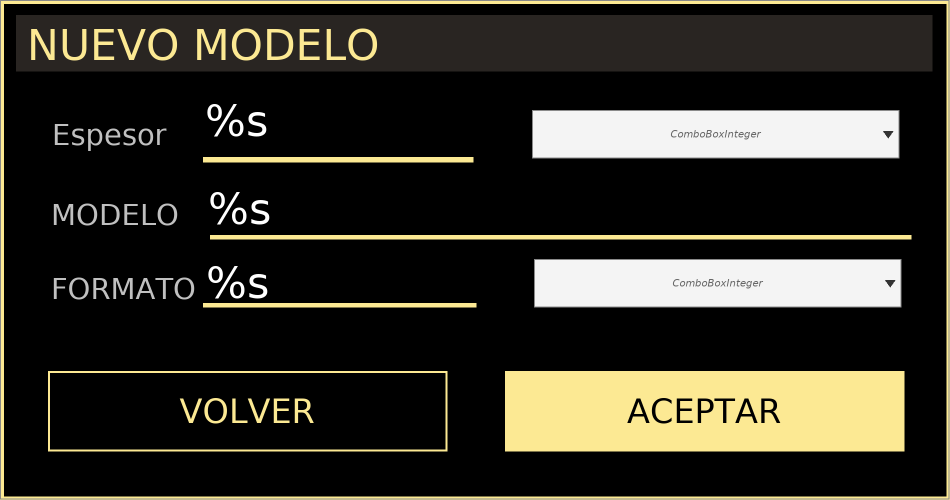
VISUALIZATION Modelo_Tabla_Ch3  // 950x500
    Rectangle (16,15 916x56)
    Rectangle (0,0 950x500)
    Label (24,17 498x56), "NUEVO MODELO"
    Rectangle (136,1125 690x58), "%s Contador piezas corte húmedo 4", text variable: FuncParoNodoRemote1CorteH2.CortHum2StrFuncParoEnviar.Cont_Piezas
    Button (871,1105 269x91), "Reset contador"
        tap FuncParoNodoLocalCorteH3.Funci_CortHum3.ResetContPiez
    ComboBoxInteger (534,259 367x48), variable: FuncParoNodoLocalCorteH3.FunGeneCortHum3.IndexListFormatoTabla, text list: 'FormatoTabla'
        p1601986498: ''
    Rectangle (205,185 701x48), "%s", text variable: FuncParoNodoLocalCorteH3.FunGeneCortHum3.s_ModeloEleccionTabla
        OnMouseDown: write the text variable via Edit
    Label (48,197 148x36), "MODELO"
    Rectangle (210,235 701x4)
    Rectangle (203,259 273x48), "%s", text variable: FuncParoNodoLocalCorteH3.sFormatoActualTabla, input disabled if: FuncParoNodoLocalCorteH3.FunGeneCortHum3.IndexListFormatoTabla<>6
        OnMouseDown: write the text variable via Edit
    Label (48,271 148x36), "FORMATO"
    Rectangle (203,303 273x4)
    Rectangle (505,371 399x80), "ACEPTAR"
        tap FuncParoNodoLocalCorteH3.FunGeneCortHum3.P_EscribirModelo
        OnMouseClick: CloseDialog Dialog=Modelo_Tabla_Ch3, Result=None, NumpadKeypadSet=True
    Rectangle (48,371 399x80), "VOLVER"
        OnMouseClick: CloseDialog Dialog=V_Emerg_Fin_Prod_Ch3, Result=None, NumpadKeypadSet=True
    Label (49,117 148x36), "Espesor"
    Rectangle (203,157 270x5)
    Rectangle (202,97 270x48), "%s", text variable: FuncParoNodoLocalCorteH3.FunGeneCortHum3.s_EspesorEleccionTabla, input disabled if: FuncParoNodoLocalCorteH3.FunGeneCortHum3.IndexListEspesorTabla<>6
        OnMouseDown: write the text variable via Edit
    ComboBoxInteger (532,110 367x48), variable: FuncParoNodoLocalCorteH3.FunGeneCortHum3.IndexListEspesorTabla, input disabled if: FuncParoNodoLocalCorteH3.FunGeneCortHum3.IndexListEspesorTabla<>6, text list: 'EspesorTabla'
        p1601986498: ''
END_VISUALIZATION

(* stored: Version 1.1.0.1, ProductVersion 3.1.4024.12
   Visu Modelo_Tabla_Ch3: Id {360bbc09-db12-451a-a31a-ee28962d287a} *)
